(* PLC project , CODESYS CODESYS V3.5 SP19 *)
(* stored: creationDateTime 2023-06-20T19:32:15.932717, modificationDateTime 2023-06-20T19:32:15.932717 *)

PROGRAM PLC_PRG_32
  VAR  (* added by the conversion: wires and edge detectors of the diagram *)
    _w58 : BOOL;
    _w72 : BOOL;
    _w80 : BOOL;
    _w91 : BOOL;
    _w102 : BOOL;
  END_VAR

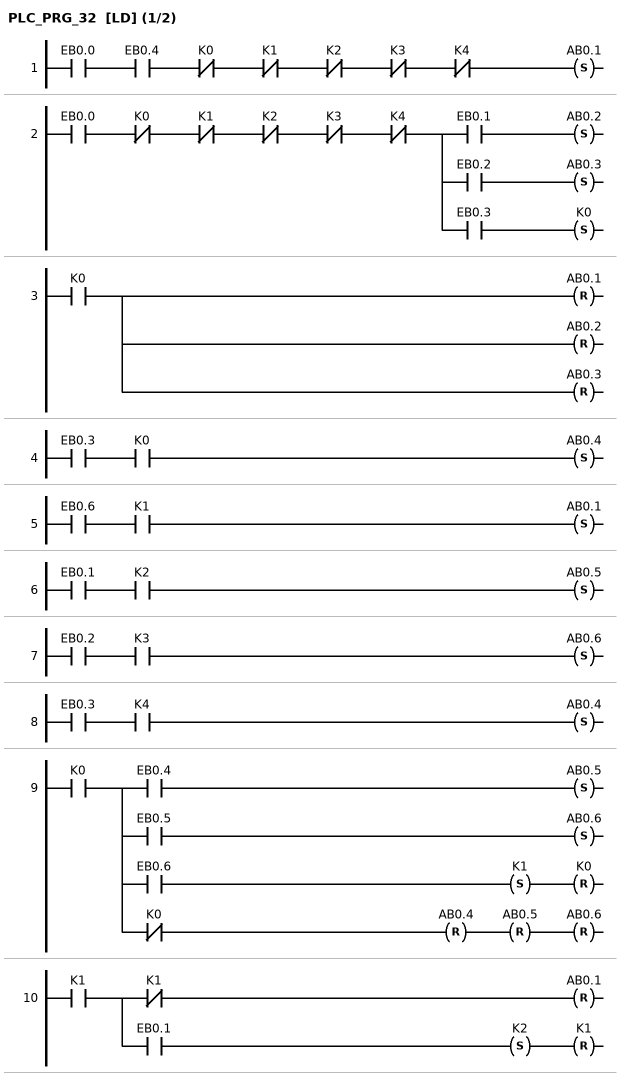
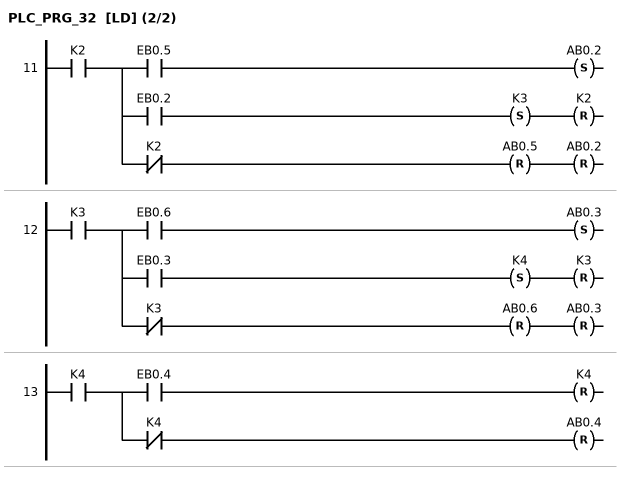
(* LD diagram, written out as Structured Text *)

IF EB0.0 AND EB0.4 AND NOT K0 AND NOT K1 AND NOT K2 AND NOT K3 AND NOT K4 THEN AB0.1 := TRUE; END_IF;

IF EB0.0 AND NOT K0 AND NOT K1 AND NOT K2 AND NOT K3 AND NOT K4 AND EB0.1 THEN AB0.2 := TRUE; END_IF;
IF EB0.0 AND NOT K0 AND NOT K1 AND NOT K2 AND NOT K3 AND NOT K4 AND EB0.2 THEN AB0.3 := TRUE; END_IF;
IF EB0.0 AND NOT K0 AND NOT K1 AND NOT K2 AND NOT K3 AND NOT K4 AND EB0.3 THEN K0 := TRUE; END_IF;

IF K0 THEN AB0.1 := FALSE; END_IF;
IF K0 THEN AB0.2 := FALSE; END_IF;
IF K0 THEN AB0.3 := FALSE; END_IF;

IF EB0.3 AND K0 THEN AB0.4 := TRUE; END_IF;

IF EB0.6 AND K1 THEN AB0.1 := TRUE; END_IF;

IF EB0.1 AND K2 THEN AB0.5 := TRUE; END_IF;

IF EB0.2 AND K3 THEN AB0.6 := TRUE; END_IF;

IF EB0.3 AND K4 THEN AB0.4 := TRUE; END_IF;

_w58 := K0;
IF _w58 AND EB0.4 THEN AB0.5 := TRUE; END_IF;
IF _w58 AND EB0.5 THEN AB0.6 := TRUE; END_IF;
IF _w58 AND EB0.6 THEN K1 := TRUE; END_IF;
IF _w58 AND EB0.6 THEN K0 := FALSE; END_IF;
IF _w58 AND NOT K0 THEN AB0.4 := FALSE; END_IF;
IF _w58 AND NOT K0 THEN AB0.5 := FALSE; END_IF;
IF _w58 AND NOT K0 THEN AB0.6 := FALSE; END_IF;

_w72 := K1;
IF _w72 AND EB0.1 THEN K2 := TRUE; END_IF;
IF _w72 AND EB0.1 THEN K1 := FALSE; END_IF;
IF _w72 AND NOT K1 THEN AB0.1 := FALSE; END_IF;

_w80 := K2;
IF _w80 AND EB0.5 THEN AB0.2 := TRUE; END_IF;
IF _w80 AND EB0.2 THEN K3 := TRUE; END_IF;
IF _w80 AND EB0.2 THEN K2 := FALSE; END_IF;
IF _w80 AND NOT K2 THEN AB0.5 := FALSE; END_IF;
IF _w80 AND NOT K2 THEN AB0.2 := FALSE; END_IF;

_w91 := K3;
IF _w91 AND EB0.6 THEN AB0.3 := TRUE; END_IF;
IF _w91 AND EB0.3 THEN K4 := TRUE; END_IF;
IF _w91 AND EB0.3 THEN K3 := FALSE; END_IF;
IF _w91 AND NOT K3 THEN AB0.6 := FALSE; END_IF;
IF _w91 AND NOT K3 THEN AB0.3 := FALSE; END_IF;

_w102 := K4;
IF _w102 AND EB0.4 THEN K4 := FALSE; END_IF;
IF _w102 AND NOT K4 THEN AB0.4 := FALSE; END_IF;
(* --- network --- *)
END_PROGRAM
